(* IEC 61131-3 sources: Industry-PLC-LLM/data/PLCBEAD_repo/PLCBEAD_PLCEmbed-main/PLC-BEAD/Source/GEB/INV, 1 file *)

(* ---- INV.ST ---- *)
FUNCTION INV:REAL

	VAR_INPUT
		X :	REAL;
	END_VAR

	IF X <> 0.0 THEN INV := 1.0 / X; END_IF;

END_FUNCTION

PROGRAM program0
	VAR
		X :	REAL;
		OUT : REAL;
	END_VAR

	OUT := INV(X);
END_PROGRAM
